(* IEC 61131-3 sources: Relay-Control-via-Modbus/pous/function-blocks, 2 files *)

(* ---- BOOL_ON_WORD.st ---- *)
FUNCTION_BLOCK BOOL_ON_WORD
VAR_INPUT
	B_IN0 : bool;
	B_IN1 : bool;
	B_IN2 : bool;
	B_IN3 : bool;
	B_IN4 : bool;
	B_IN5 : bool;
	B_IN6 : bool;
	B_IN7 : bool;
	B_IN8 : bool;
	B_IN9 : bool;
	B_IN10 : bool;
	B_IN11 : bool;
	B_IN12 : bool;
	B_IN13 : bool;
	B_IN14 : bool;
	B_IN15 : bool;
END_VAR

VAR_OUTPUT
	WORD_OUT : word;
END_VAR

WORD_OUT := 0;
IF B_IN0  THEN WORD_OUT := WORD_OUT OR 16#0001; END_IF;
IF B_IN1  THEN WORD_OUT := WORD_OUT OR 16#0002; END_IF;
IF B_IN2  THEN WORD_OUT := WORD_OUT OR 16#0004; END_IF;
IF B_IN3  THEN WORD_OUT := WORD_OUT OR 16#0008; END_IF;
IF B_IN4  THEN WORD_OUT := WORD_OUT OR 16#0010; END_IF;
IF B_IN5  THEN WORD_OUT := WORD_OUT OR 16#0020; END_IF;
IF B_IN6  THEN WORD_OUT := WORD_OUT OR 16#0040; END_IF;
IF B_IN7  THEN WORD_OUT := WORD_OUT OR 16#0080; END_IF;
IF B_IN8  THEN WORD_OUT := WORD_OUT OR 16#0100; END_IF;
IF B_IN9  THEN WORD_OUT := WORD_OUT OR 16#0200; END_IF;
IF B_IN10 THEN WORD_OUT := WORD_OUT OR 16#0400; END_IF;
IF B_IN11 THEN WORD_OUT := WORD_OUT OR 16#0800; END_IF;
IF B_IN12 THEN WORD_OUT := WORD_OUT OR 16#1000; END_IF;
IF B_IN13 THEN WORD_OUT := WORD_OUT OR 16#2000; END_IF;
IF B_IN14 THEN WORD_OUT := WORD_OUT OR 16#4000; END_IF;
IF B_IN15 THEN WORD_OUT := WORD_OUT OR 16#8000; END_IF;

END_FUNCTION_BLOCK

(* ---- WORD_ON_BOOL.st ---- *)
FUNCTION_BLOCK WORD_ON_BOOL
VAR_INPUT
	WORD_IN : word;
END_VAR

VAR_OUTPUT
	B_OUT0 : bool;
	B_OUT1 : bool;
	B_OUT2 : bool;
	B_OUT3 : bool;
	B_OUT4 : bool;
	B_OUT5 : bool;
	B_OUT6 : bool;
	B_OUT7 : bool;
	B_OUT8 : bool;
	B_OUT9 : bool;
	B_OUT10 : bool;
	B_OUT11 : bool;
	B_OUT12 : bool;
	B_OUT13 : bool;
	B_OUT14 : bool;
	B_OUT15 : bool;
END_VAR

B_OUT0  := (WORD_IN AND 16#0001) <> 0;
B_OUT1  := (WORD_IN AND 16#0002) <> 0;
B_OUT2  := (WORD_IN AND 16#0004) <> 0;
B_OUT3  := (WORD_IN AND 16#0008) <> 0;
B_OUT4  := (WORD_IN AND 16#0010) <> 0;
B_OUT5  := (WORD_IN AND 16#0020) <> 0;
B_OUT6  := (WORD_IN AND 16#0040) <> 0;
B_OUT7  := (WORD_IN AND 16#0080) <> 0;
B_OUT8  := (WORD_IN AND 16#0100) <> 0;
B_OUT9  := (WORD_IN AND 16#0200) <> 0;
B_OUT10 := (WORD_IN AND 16#0400) <> 0;
B_OUT11 := (WORD_IN AND 16#0800) <> 0;
B_OUT12 := (WORD_IN AND 16#1000) <> 0;
B_OUT13 := (WORD_IN AND 16#2000) <> 0;
B_OUT14 := (WORD_IN AND 16#4000) <> 0;
B_OUT15 := (WORD_IN AND 16#8000) <> 0;

END_FUNCTION_BLOCK
